FUNCTION_BLOCK "LEXCHANGETRAY_U2Em1SingleTM"
TITLE = EXCHANGETRAY_U2Em1SingleTM
{ S7_Optimized_Access := 'TRUE' ; Published := 'TRUE' }
AUTHOR : 'SUP/Zhang Shi Long'
FAMILY : SUP
VERSION : 0.1
//Exchange Tray function
   VAR_INPUT
      trayAutomaticDischargeDetectionEm1 { ExternalAccessible := 'False'; ExternalVisible := 'False'; ExternalWritable := 'False'} : Bool;   // Tray automatic discharge detection sensor EM1
      trayAutomaticFeedingDetectionEm1 { ExternalAccessible := 'False'; ExternalVisible := 'False'; ExternalWritable := 'False'} : Bool;   // Tray automatic feeding detection sensor EM1
      restraintTrayAntiReverseDetection2Em1 { ExternalAccessible := 'False'; ExternalVisible := 'False'; ExternalWritable := 'False'} : Bool;   // Restraint tray anti-reverse detection sensor 2 EM1
      restraintTrayAntiReverseDetection1Em1 { ExternalAccessible := 'False'; ExternalVisible := 'False'; ExternalWritable := 'False'} : Bool;   // Restraint tray anti-reverse detection sensor 1 EM1
   END_VAR

   VAR_IN_OUT
      configuration : "LEXCHANGETRAY_typeRollerIoSignalConfigeration";   // Configuration parameters for tray module
      moduleInterface : "LEXCHANGETRAY_typeRollerIoSignalInterface";   // Module interface for tray control
      controlNode : "LEXCHANGETRAY_typeRollerIoSignalControlNode";   // Control node parameters
   END_VAR

   VAR
      statManualCommands { S7_SetPoint := 'False'} : "LEXCHANGETRAY_typeRollerIoSignalManualCommands";   // Manual commands execution status
      statProcessValues { S7_SetPoint := 'False'} : "LEXCHANGETRAY_typeRollerIoSignalProcessValues";   // Process values monitoring status
      statDiagnostics : "LBC_typeDiagnostics";   // Diagnostics information status
      statSimActive : Bool;   // Simulation mode active status
      statSimActivePrevious : Bool;   // Previous simulation mode status
      statFbState : Word;   // Current function block state
      statFbStatePrevious : Word;   // Previous function block state
   END_VAR

   VAR_TEMP
      tempSimActiveEdge : Bool;
   END_VAR


BEGIN
	REGION BLOCK INFO HEADER
	    //===============================================================================
	    // Siemens / (c)Copyright 2020-2024
	    //-------------------------------------------------------------------------------
	    // Title:            Roller Simulation Signal Processing Module
	    // 标题:             滚筒模拟信号处理模块
	    // Comment/Function: This module is responsible for processing input signals related to Roller simulation,
	    //                    mapping different input sources according to the simulation activation status,
	    //                    resetting relevant signals, and outputting processed data.
	    // 注释/功能:        此模块负责处理与 滚筒模拟相关的输入信号，
	    //                    根据模拟激活状态映射不同输入源，
	    //                    重置相关信号，并输出处理后的数据。
	    // Library/Family:   EXCHANGETRAY - Library of Basic
	    // 库/家族:         换盘机 - 基本控制模块库
	    // Author:           Siemens Digital Industries
	    // 作者:            西门子数字工业
	    // Tested with:      S7-PLCSIM Advanced 6.0
	    // 测试环境:        S7-PLCSIM Advanced 6.0
	    // Engineering:      TIA Portal V19
	    // 工程环境:        TIA Portal V19
	    // Restrictions:     ENO mechanism is not used - forced to False.
	    // 限制条件:        不使用 ENO 机制 - 强制设置为 False。
	    // Requirements:     PLC (S7-1200 / S7-1500)
	    // 要求:            PLC (S7-1200 / S7-1500)
	    //-------------------------------------------------------------------------------
	    // Change log table:
	    // Version  | Date       | Expert in charge        | Changes applied
	    //----------|------------|-------------------------|-----------------------------
	    // 01.00.00 | 17.04.2025 | SIMATIC Systems Support | Updated block info and comments following AIupdate.scl style.
	    // 版本     | 日期       | 负责人                  | 更改内容
	    //----------|------------|-------------------------|-----------------------------
	    // 01.00.00 | 2025年4月17日 | SIMATIC系统支持        | 参照 LBC 风格更新块信息和注释。
	    //===============================================================================
	END_REGION BLOCK INFO HEADER

	REGION DESCRIPTION
	    (/*
	    This module processes input signals related to the Roller simulation.
	    It checks whether the simulation mode is active based on the configuration.
	    When the simulation is active, it combines the manual commands and real input signals;
	    otherwise, it directly uses the real input signals.
	    Additionally, it resets relevant manual commands when the simulation is inactive
	    and finally outputs the processed data to the module interface and control node.

	    此模块处理与 滚筒模拟相关的输入信号。
	    它根据配置检查模拟模式是否激活。
	    当模拟激活时，它将手动命令和真实输入信号进行组合；
	    否则，它直接使用真实输入信号。
	    此外，当模拟未激活时，它会重置相关的手动命令，
	    最后将处理后的数据输出到模块接口和控制节点。
	    */)
	END_REGION DESCRIPTION

	REGION INITIALISATION
	    // Reset relevant manual commands when the simulation is inactive
	    // 模拟未激活时，重置相关的手动命令
	    IF NOT #statSimActive OR (#controlNode.reset) THEN
	        #controlNode.reset :=
	        #statManualCommands.trayAutomaticDischargeDetectionEm1 := FALSE;
	        #statManualCommands.trayAutomaticFeedingDetectionEm1 := FALSE;
	        #statManualCommands.restraintTrayAntiReverseDetection2Em1 := FALSE;
	        #statManualCommands.restraintTrayAntiReverseDetection1Em1 := FALSE;
	    END_IF;
	END_REGION INITIALISATION

	REGION PROGRAM LOGIC
	    REGION PROCESS INPUT SIGNALS
	        REGION Input configuration parameter
	            // Assign the simulation activation status from the configuration to the static variable
	            // 将配置中的模拟激活状态赋值给静态变量
	            #statSimActive := #configuration.simActive;
	        END_REGION
	        // Map the commands from the module interface to the manual commands
	        // 将模块接口的命令映射到手动命令
	        #statManualCommands := #moduleInterface.commands;

	        // Map input signals based on the simulation activation status
	        // 根据模拟激活状态映射输入信号
	        IF #statSimActive THEN
	            // Combine manual commands and real input signals when simulation is active
	            // 模拟激活时，组合手动命令和真实输入信号
	            #statProcessValues.trayAutomaticDischargeDetectionEm1 := #statManualCommands.trayAutomaticDischargeDetectionEm1 OR #trayAutomaticDischargeDetectionEm1;
	            #statProcessValues.trayAutomaticFeedingDetectionEm1 := #statManualCommands.trayAutomaticFeedingDetectionEm1 OR #trayAutomaticFeedingDetectionEm1;
	            #statProcessValues.restraintTrayAntiReverseDetection2Em1 := #statManualCommands.restraintTrayAntiReverseDetection2Em1 OR #restraintTrayAntiReverseDetection2Em1;
	            #statProcessValues.restraintTrayAntiReverseDetection1Em1 := #statManualCommands.restraintTrayAntiReverseDetection1Em1 OR #restraintTrayAntiReverseDetection1Em1;
	        ELSE
	            // Use real input signals directly when simulation is inactive
	            // 模拟未激活时，直接使用真实输入信号
	            #statProcessValues.trayAutomaticDischargeDetectionEm1 := #trayAutomaticDischargeDetectionEm1;
	            #statProcessValues.trayAutomaticFeedingDetectionEm1 := #trayAutomaticFeedingDetectionEm1;
	            #statProcessValues.restraintTrayAntiReverseDetection2Em1 := #restraintTrayAntiReverseDetection2Em1;
	            #statProcessValues.restraintTrayAntiReverseDetection1Em1 := #restraintTrayAntiReverseDetection1Em1;
	        END_IF;

	        REGION SIMULATE MODE
	            // Simulation mode logic can be added here
	            // 模拟模式逻辑可在此处添加
	        END_REGION SIMULATE MODE
	        REGION Interlock dependent edge commands
	            // Detect the rising edge of the simulation activation signal
	            // 检测模拟激活信号的上升沿
	            #tempSimActiveEdge := #statSimActive AND NOT #statSimActivePrevious;
	        END_REGION Interlock dependent edge commands
	    END_REGION PROCESS INPUT SIGNALS
	END_REGION PROGRAM LOGIC

	REGION OUTPUTS
	    // Assign the simulation activation status to the monitoring structure
	    // 将模拟激活状态赋值给监控结构
	    #statProcessValues.simulated := #statSimActive;
	    // Write the manual commands to the module interface
	    // 将手动命令写入模块接口
	    #moduleInterface.commands := #statManualCommands;
	    // Write the process values to the module interface monitoring
	    // 将过程值写入模块接口监控
	    #moduleInterface.monitoring := #statProcessValues;
	    // Write the simulation status and processed signals to the control node monitoring
	    // 将模拟状态和处理后的信号写入控制节点监控
	    #controlNode.monitoring.simulated := #statProcessValues.simulated;
	    #controlNode.monitoring.trayAutomaticDischargeDetectionEm1 := #statProcessValues.trayAutomaticDischargeDetectionEm1;
	    #controlNode.monitoring.trayAutomaticFeedingDetectionEm1 := #statProcessValues.trayAutomaticFeedingDetectionEm1;
	    #controlNode.monitoring.restraintTrayAntiReverseDetection2Em1 := #statProcessValues.restraintTrayAntiReverseDetection2Em1;
	    #controlNode.monitoring.restraintTrayAntiReverseDetection1Em1 := #statProcessValues.restraintTrayAntiReverseDetection1Em1;
	    // ENO mechanism disabled, ENO - forced to False
	    // ENO 机制禁用，强制设置为 False
	    ENO := False;
	END_REGION OUTPUTS

END_FUNCTION_BLOCK

